(* IEC 61131-3 sources: repolevel_ST_code_completion/dataset/generation_context_ground_truth/elevator, 5 files *)

(* ---- F_DetectCurrentFloor.st ---- *)
// 根据传感器输入确定当前楼层
IF FloorSensor0 THEN
	F_DetectCurrentFloor := 0;
ELSIF FloorSensor1 THEN
	F_DetectCurrentFloor := 1;
ELSIF FloorSensor2 THEN
	F_DetectCurrentFloor := 2;
ELSIF FloorSensor3 THEN
	F_DetectCurrentFloor := 3;
ELSE
	// 没有传感器信号时，保持当前楼层
	F_DetectCurrentFloor := CurrentFloor;
END_IF

(* ---- F_RegisterCalls.st ---- *)
// 注册各楼层的呼叫请求
IF CallGround THEN
	TargetFloors[0] := TRUE;
END_IF

IF CallFloor1 THEN
	TargetFloors[1] := TRUE;
END_IF

IF CallFloor2 THEN
	TargetFloors[2] := TRUE;
END_IF

IF CallFloor3 THEN
	TargetFloors[3] := TRUE;
END_IF

(* ---- F_UpdateDoorAnimation.st ---- *)
VAR
	nNewAni			:	DINT;		// 新的动画值
END_VAR

nNewAni := nCurrentAni;

// 开门动画（增加动画值）
IF bOpenDoor AND nNewAni < nMaxAni AND bCallFloor THEN
	nNewAni := nNewAni + 1;
END_IF

// 关门动画（减少动画值）
IF bCloseDoor AND nNewAni > 0 THEN
	nNewAni := nNewAni - 1;
END_IF

F_UpdateDoorAnimation := nNewAni;

(* ---- FB_ElevatorDoorController.st ---- *)
VAR
	fbDoorTimer			:	TON;		// 开门延时定时器
	fbCloseDoorTimer	:	TON;		// 关门延时定时器
	nState				:	INT;		// 状态机
END_VAR

CASE nState OF
	0: // 空闲状态
		bOpenDoor := FALSE;
		bCloseDoor := FALSE;
		bDoorReady := TRUE;

		IF bArrivedAtTarget THEN
			nState := 1; // 开始开门流程
		END_IF

	1: // 开门延时
		bCloseDoor := FALSE;
		bDoorReady := FALSE;
		fbDoorTimer(IN := TRUE, PT := T#2S);

		IF fbDoorTimer.Q THEN
			fbDoorTimer(IN := FALSE);
			nState := 2;
		END_IF

	2: // 开门
		bOpenDoor := TRUE;
		bDoorOpen := TRUE;
		nState := 3;

	3: // 等待开始关门
		IF NOT bArrivedAtTarget THEN
			nState := 4; // 开始关门流程
		END_IF

	4: // 关门
		bOpenDoor := FALSE;
		bCloseDoor := TRUE;
		bDoorOpen := FALSE;
		fbCloseDoorTimer(IN := TRUE, PT := T#2S);

		IF fbCloseDoorTimer.Q AND bDoorClosed THEN
			fbCloseDoorTimer(IN := FALSE);
			nState := 0; // 返回空闲
		END_IF
END_CASE

(* ---- FB_ElevatorMovement.st ---- *)
VAR
	fbMoveDelayTimer	:	TON;				// 移动延时定时器
	i					:	INT;				// 循环变量
	bHasUpperRequest	:	BOOL;				// 有更高楼层请求
	bHasLowerRequest	:	BOOL;				// 有更低楼层请求
END_VAR

// 检查是否到达目标楼层
IF TargetFloors[CurrentFloor] THEN
	bArrivedAtTarget := TRUE;
	TargetFloors[CurrentFloor] := FALSE; // 清除请求
	bMovingUp := FALSE;
	bMovingDown := FALSE;
	RETURN;
ELSE
	bArrivedAtTarget := FALSE;
END_IF

// 只有门准备好才能移动
IF NOT bDoorReady THEN
	RETURN;
END_IF

// 检查是否有更高楼层的请求
bHasUpperRequest := FALSE;
FOR i := CurrentFloor + 1 TO 3 DO
	IF TargetFloors[i] THEN
		bHasUpperRequest := TRUE;
		EXIT;
	END_IF
END_FOR

// 检查是否有更低楼层的请求
bHasLowerRequest := FALSE;
FOR i := CurrentFloor - 1 TO 0 BY -1 DO
	IF TargetFloors[i] THEN
		bHasLowerRequest := TRUE;
		EXIT;
	END_IF
END_FOR

// 移动逻辑
IF bMovingUp OR (NOT bMovingDown AND bHasUpperRequest) THEN
	// 向上移动
	IF bHasUpperRequest THEN
		fbMoveDelayTimer(IN := TRUE, PT := T#500MS);
		IF fbMoveDelayTimer.Q THEN
			bMovingUp := TRUE;
			bMovingDown := FALSE;
			fbMoveDelayTimer(IN := FALSE);
		END_IF
	ELSE
		// 没有更高请求，改变方向
		bMovingUp := FALSE;
		IF bHasLowerRequest THEN
			bMovingDown := TRUE;
		END_IF
	END_IF
ELSIF bMovingDown OR (NOT bMovingUp AND bHasLowerRequest) THEN
	// 向下移动
	IF bHasLowerRequest THEN
		fbMoveDelayTimer(IN := TRUE, PT := T#500MS);
		IF fbMoveDelayTimer.Q THEN
			bMovingDown := TRUE;
			bMovingUp := FALSE;
			fbMoveDelayTimer(IN := FALSE);
		END_IF
	ELSE
		// 没有更低请求，改变方向
		bMovingDown := FALSE;
		IF bHasUpperRequest THEN
			bMovingUp := TRUE;
		END_IF
	END_IF
ELSE
	// 初始状态，默认向上
	IF bHasUpperRequest THEN
		bMovingUp := TRUE;
	ELSIF bHasLowerRequest THEN
		bMovingDown := TRUE;
	END_IF
END_IF
